// SIMATIC S7-200 project (STEP 7-Micro/WIN), CPU 221 REL 01.10

ORGANIZATION_BLOCK MAIN:OB1
TITLE=
BEGIN
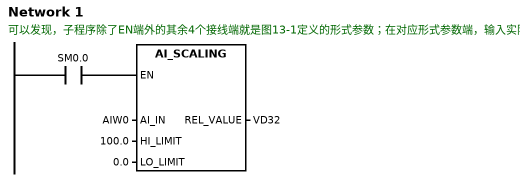
Network 1
// 可以发现，子程序除了EN端外的其余4个接线端就是图13-1定义的形式参数；在对应形式参数端，输入实际参数AIW0，模拟量上下限100度和0度，以及模拟量转换的保存地址VD32
// (network saved uncompiled; LAD cells follow)
// row 0: c0 -| |- SM0.0  c1 [AI_SCALING EN:=power@row0, AI_IN:=AIW0, HI_LIMIT:=100.0, LO_LIMIT:=0.0, REL_VALUE=>VD32]
// row 1: c1 [box]
END_ORGANIZATION_BLOCK

SUBROUTINE_BLOCK AI_SCALING:SBR0
TITLE=
VAR_INPUT
AI_IN:INT;	// LW0 模拟输入
HI_LIMIT:REAL;	// LD2 模拟输入对应的实际工程量的上限
LO_LIMIT:REAL;	// LD6 模拟输入对应的实际工程量的下限
END_VAR
VAR_OUTPUT
REL_VALUE:REAL;	// LD10 转换后的实际工程值
END_VAR
BEGIN
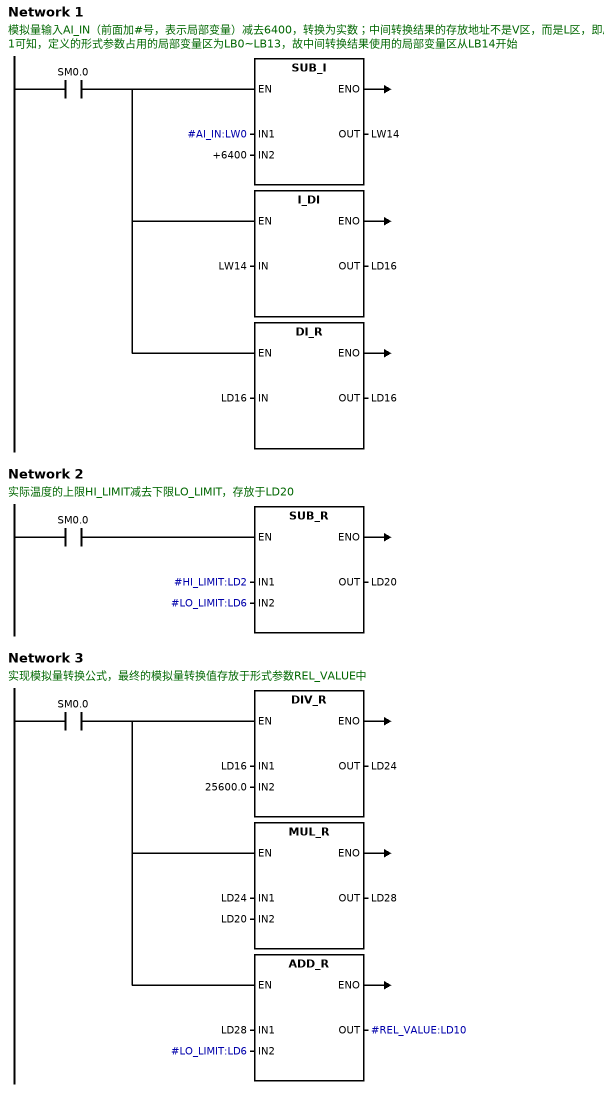
Network 1
// 模拟量输入AI_IN（前面加#号，表示局部变量）减去6400，转换为实数；中间转换结果的存放地址不是V区，而是L区，即局部变量区；由图13-1可知，定义的形式参数占用的局部变量区为LB0~LB13，故中间转换结果使用的局部变量区从LB14开始
LD     SM0.0
MOVW   #AI_IN:LW0, LW14
-I     +6400, LW14
ITD    LW14, LD16
DTR    LD16, LD16
Network 2
// 实际温度的上限HI_LIMIT减去下限LO_LIMIT，存放于LD20
LD     SM0.0
MOVR   #HI_LIMIT:LD2, LD20
-R     #LO_LIMIT:LD6, LD20
Network 3
// 实现模拟量转换公式，最终的模拟量转换值存放于形式参数REL_VALUE中
LD     SM0.0
MOVR   LD16, LD24
/R     25600.0, LD24
MOVR   LD24, LD28
*R     LD20, LD28
MOVR   LD28, #REL_VALUE:LD10
+R     #LO_LIMIT:LD6, #REL_VALUE:LD10
END_SUBROUTINE_BLOCK
